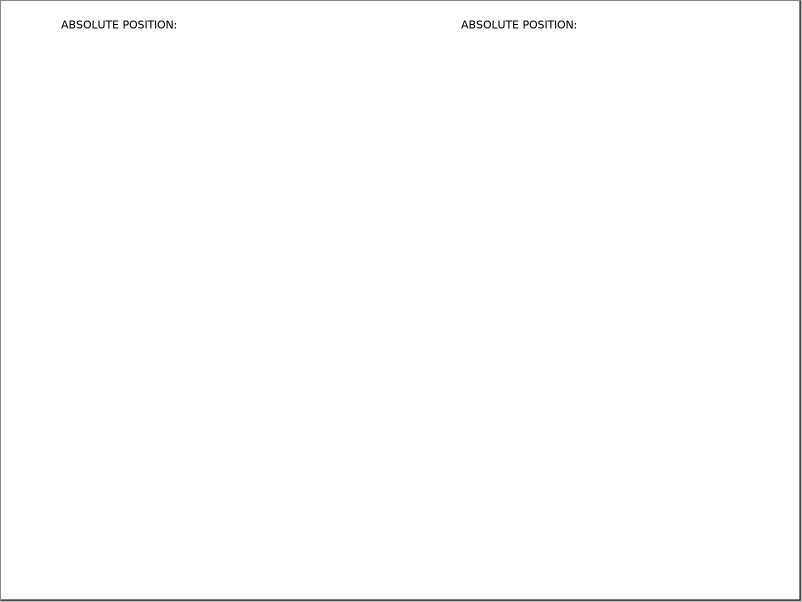
VISUALIZATION F41_Gear_In_Dynamic  // 802x602
    Rectangle (0,0 800x600)
    Label (10,10 170x30), "ABSOLUTE POSITION:"
    Label (410,10 170x30), "ABSOLUTE POSITION:"
END_VISUALIZATION

(* stored: Version 1.1.0.1, ProductVersion 3.1.4022.7
   Visu F41_Gear_In_Dynamic: Id {65ee6377-6b0a-400b-bd12-f8274c44d409} *)
